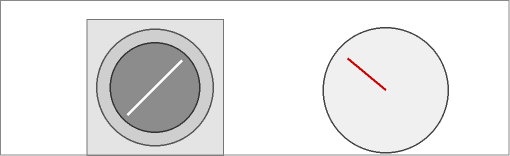
VISUALIZATION Visualization  // 510x156
    Potentiometer360 (77,19 156x137), variable: MAIN.velocity, style: Potentiometer-Potentiometer360-Gray, scale format: %.1f, scale 0..1
        p2431819421: Outside
    Meter180 (261,27 249x126), value: MAIN.PosPiston, style: Meter-Meter180-Gray, scale format: %.1f, scale 25..65
        p518627256: mm
END_VISUALIZATION

(* stored: Version 1.1.0.1, ProductVersion 3.1.4024.10
   Visu Visualization: Id {60b7cc59-b549-4590-9a54-d91f4387e167} *)
